TYPE Inbound :
STRUCT
	roller	: Roller;
	photo_sensor_mute	 : BOOL;
	photo_sensor	: BOOL;
END_STRUCT
END_TYPE

(* stored: Version 1.1.0.1, ProductVersion 3.1.4024.12
   DUT Inbound: Id {3c45f76f-b107-4a7f-8658-42ef4037bda9} *)
